// TIA Portal V20 export
DATA_BLOCK "Instance_FB_Digital_Input_DB"   // DB101
// stored: AutoNumber false, InstanceOfName FB_Digital_Input, InstanceOfType FB
"FB_Digital_Input"
   // VAR_INPUT
   //    DI_Emergency_Stop_Release : Bool;
   //    DI_Sensor_Water_Fountain_Before_Entrace_Functional_Test_Spinner_Conveyor_Belt : Bool;
   //    DI_Sensor_Water_Fountain_Entrace_Functional_Test_Spinner_Conveyor_Belt : Bool;
   //    DI_Sensor_Water_Fountain_Entrace_Functional_Test_After_Spinner_Conveyor_Belt : Bool;
   //    DI_Trigger_Read_Serial_Number_Entrace_Functional_Test : Bool;
   //    DI_Sensor_Water_Fountain_Geting_Exit_Rework_Conveyor_Belt : Bool;
   //    DI_Button_Water_Fountain_Get_Exit_Rework_Conveyor_Belt : Bool;
   //    DI_Trigger_Read_Serial_Number_Exit_Functional_Test : Bool;
   //    DI_Sensor_Water_Fountain_Exit_Functional_Test_Spinner_Conveyor_Belt : Bool;
   //    DI_Sensor_Water_Fountain_Exit_Functional_Test_After_Spinner_Conveyor_Belt : Bool;
   //    DI_Sensor_Water_Fountain_Geting_Entrace_Rework_Conveyor_Belt_Start : Bool;
   //    DI_Sensor_Water_Fountain_Geting_Entrace_Rework_Conveyor_Belt_Finish : Bool;
   //    DI_Carousel_Frequency_Inverter_Fail : Bool;
   //    DI_Conveyor_Belt_Functional_Test_Inverter_Fail : Bool;
   //    DI_Selected_Voltage_220V : Bool;
   //    DI_Selected_Voltage_127V : Bool;
   //    DI_Sensor_Spinner_Entrace_Functional_Test_Position_Withdrawn : Bool;
   //    DI_Sensor_Spinner_Entrace_Functional_Test_Position_Advanced : Bool;
   //    DI_Sensor_Spinner_Exit_Functional_Test_Position_Withdrawn : Bool;
   //    DI_Sensor_Spinner_Exit_Functional_Test_Position_Advanced : Bool;
   //    DI_Digital_Input_20 : Bool;
   //    DI_Digital_Input_21 : Bool;
   //    DI_Digital_Input_22 : Bool;
   //    DI_Digital_Input_23 : Bool;
   //    DI_Digital_Input_24 : Bool;
   //    DI_Digital_Input_25 : Bool;
   //    DI_Digital_Input_26 : Bool;
   //    DI_Digital_Input_27 : Bool;
   //    DI_Digital_Input_28 : Bool;
   //    DI_Digital_Input_29 : Bool;
   // END_VAR
   // VAR_OUTPUT
   //    DB_Emergency_Stop_Release : Bool;
   //    DB_Sensor_Water_Fountain_Before_Entrace_Functional_Test_Spinner_Conveyor_Belt : Bool;
   //    DB_Sensor_Water_Fountain_Entrace_Functional_Test_Spinner_Conveyor_Belt : Bool;
   //    DB_Sensor_Water_Fountain_Entrace_Functional_Test_After_Spinner_Conveyor_Belt : Bool;
   //    DB_Trigger_Read_Serial_Number_Entrace_Functional_Test : Bool;
   //    DB_Sensor_Water_Fountain_Geting_Exit_Rework_Conveyor_Belt : Bool;
   //    DB_Button_Water_Fountain_Get_Exit_Rework_Conveyor_Belt : Bool;
   //    DB_Trigger_Read_Serial_Number_Exit_Functional_Test : Bool;
   //    DB_Sensor_Water_Fountain_Exit_Functional_Test_Spinner_Conveyor_Belt : Bool;
   //    DB_Sensor_Water_Fountain_Exit_Functional_Test_After_Spinner_Conveyor_Belt : Bool;
   //    DB_Sensor_Water_Fountain_Geting_Entrace_Rework_Conveyor_Belt_Start : Bool;
   //    DB_Sensor_Water_Fountain_Geting_Entrace_Rework_Conveyor_Belt_Finish : Bool;
   //    DB_Carousel_Frequency_Inverter_Fail : Bool;
   //    DB_Conveyor_Belt_Functional_Test_Inverter_Fail : Bool;
   //    DB_Selected_Voltage_220V : Bool;
   //    DB_Selected_Voltage_127V : Bool;
   //    DB_Sensor_Spinner_Entrace_Functional_Test_Position_Withdrawn : Bool;
   //    DB_Sensor_Spinner_Entrace_Functional_Test_Position_Advanced : Bool;
   //    DB_Sensor_Spinner_Exit_Functional_Test_Position_Withdrawn : Bool;
   //    DB_Sensor_Spinner_Exit_Functional_Test_Position_Advanced : Bool;
   //    DB_Digital_Input_20 : Bool;
   //    DB_Digital_Input_21 : Bool;
   //    DB_Digital_Input_22 : Bool;
   //    DB_Digital_Input_23 : Bool;
   //    DB_Digital_Input_24 : Bool;
   //    DB_Digital_Input_25 : Bool;
   //    DB_Digital_Input_26 : Bool;
   //    DB_Digital_Input_27 : Bool;
   //    DB_Digital_Input_28 : Bool;
   //    DB_Digital_Input_29 : Bool;
   // END_VAR
BEGIN
END_DATA_BLOCK
